PROGRAM AnalogConversion
VAR
	
	i					: INT := 1; //charger 1-8
	j					: INT := 1;  // section 1 - 4 
	k					: INT := 1;  // cap 1-10
	m					: INT := 1; //form cap 1-12

END_VAR

//Converting raw data into Voltage Reading (0-10V), (0.5-4.5V)   
//unfinish


//MCP Charger 
//Analog Input
FOR i := 1 TO 8 BY 1 DO
	
	MCP_IO.Charger[i].ChargerType_12kV := NOT MCP_IO.Charger[i].ChargerType_50kV;
	//50kV chargers feedback
	MCP_IO.Charger[i].voltageFeedback_norm := Norm_x (raw_input := INT_TO_REAL (MCP_IO.Charger[i].voltageFeedback_raw),
													x_max := 32767,
													x_min := 0);

	MCP_IO.Charger[i].voltageFeedback := (EngVal.Max_50kVChargerVoltage - EngVal.Min_50kVChargerVoltage) * ADC_10V(
																							normal_input := MCP_IO.Charger[i].voltageFeedback_norm,
																							x_max := 10,
																							x_min := 0);
												
	MCP_IO.Charger[i].currentFeedback_norm := Norm_x (raw_input := INT_TO_REAL (MCP_IO.Charger[i].currentFeedback_raw),
													x_max := 32767,
													x_min := 0);

	MCP_IO.Charger[i].currentFeedback := (EngVal.Max_50kVChargerCurrent - EngVal.Min_50kVChargerCurrent) * ADC_10V(
																							normal_input := MCP_IO.Charger[i].currentFeedback_norm,
																							x_max := 10,
																							x_min := 0);
	//12kV chargers ???
	
	
END_FOR;

//Analog Output
//voltageSP = Required Charge Voltage******************
FOR i := 1 TO 8 BY 1 DO
	
	//if 50kV config selected
	IF MCP_IO.Charger[i].ChargerType_50kV = TRUE THEN 
		//set limits of charger voltage input 
		IF MCP_IO.Charger[i].voltageSP >= REAL_TO_INT (EngVal.Max_50kVChargerVoltage) THEN
			MCP_IO.Charger[i].voltageSP := REAL_TO_INT (EngVal.Max_50kVChargerVoltage);
		END_IF;
		
	//prepare output signal for 50kV chargers.
		MCP_IO.Charger[i].voltageSP_norm := Norm_x (raw_input := INT_TO_REAL (MCP_IO.Charger[i].voltageSP), 
												x_max := EngVal.Max_50kVChargerVoltage,
												x_min := EngVal.Min_50kVChargerVoltage);	
												
		MCP_IO.Charger[i].voltageSP_raw := AQ (norm_input := MCP_IO.Charger[i].voltageSP_norm, 
												x_max := 10,
												x_min := 0);
		
	END_IF;
		
	//if 12kV config selected
	IF MCP_IO.Charger[i].ChargerType_12kV = TRUE THEN
		//set limits of charger voltage input 
		IF MCP_IO.Charger[i].voltageSP >= REAL_TO_INT (EngVal.Max_12kVChargerVoltage) THEN
			MCP_IO.Charger[i].voltageSP := REAL_TO_INT (EngVal.Max_12kVChargerVoltage);
		END_IF;
		
		
		//prepare output signal for 12kV chargers.
		MCP_IO.Charger[i].voltageSP_norm := Norm_x (raw_input := INT_TO_REAL (MCP_IO.Charger[i].voltageSP), 
												x_max := EngVal.Max_12kVChargerVoltage,
												x_min := EngVal.Min_12kVChargerVoltage);
		
		MCP_IO.Charger[i].voltageSP_raw := AQ (norm_input := MCP_IO.Charger[i].voltageSP_norm, 
												x_max := 10,
												x_min := 0); 
	END_IF;	
												
	//limite for output sigal (<= 10V)  this should not happen
	IF MCP_IO.Charger[i].voltageSP_raw >= 32767 THEN 
		MCP_IO.Charger[i].voltageSP_raw := 32767; 										
	END_IF;
	
END_FOR;

//prepare analog output for gls chargers.	
MCP_IO.GLS1_voltageSP_norm := Norm_x (raw_input := INT_TO_REAL (MCP_IO.GLS1_voltageSP),
									x_max := EngVal.Max_GLS1_ChargerV,
									x_min := 0);
MCP_IO.GLS1_voltageSP_raw:= AQ (norm_input := MCP_IO.GLS1_voltageSP_norm,
									x_max := 10,
									x_min := 0);									
									
MCP_IO.GLS2_voltageSP_norm := Norm_x (raw_input := INT_TO_REAL (MCP_IO.GLS2_voltageSP),
									x_max := EngVal.Max_GLS2_ChargerV,
									x_min := 0);
MCP_IO.GLS2_voltageSP_raw:= AQ (norm_input := MCP_IO.GLS2_voltageSP_norm,
									x_max := 10,
									x_min := 0);	

MCP_IO.GLS3_voltageSP_norm := Norm_x (raw_input := INT_TO_REAL (MCP_IO.GLS3_voltageSP),
									x_max := EngVal.Max_GLS3_ChargerV,
									x_min := 0);
MCP_IO.GLS3_voltageSP_raw:= AQ (norm_input := MCP_IO.GLS3_voltageSP_norm,
									x_max := 10,
									x_min := 0);	

//LCP 1 - 3 AI
FOR j := 1 TO 3 BY 1 DO 
	FOR k := 1 TO 10 BY 1 DO 
		LCP.Section[j].Peak.Cap[k].voltageFeedback_Norm := Norm_x (raw_input := INT_TO_REAL (LCP.Section[j].Peak.Cap[k].voltageFeedback_raw),
																x_max := 32767,
																x_min := 0);
																
		LCP.Section[j].Peak.Cap[k].voltageFeedback := (EngVal.Max_CapVoltage - EngVal.Min_CapVoltage) * ADC_10V (
																								normal_input := LCP.Section[j].Peak.Cap[k].voltageFeedback_Norm,
																								x_max := 10,
																								x_min := 0);
		//sustain caps 1 - 2
		LCP.Section[j].Sust.Cap[1].voltageFeedback_Norm := Norm_x (raw_input := INT_TO_REAL (LCP.Section[j].Sust.Cap[1].voltageFeedback_raw),
																x_max := 32767,
																x_min := 0);
																
		LCP.Section[j].Sust.Cap[1].voltageFeedback := (EngVal.Max_CapVoltage - EngVal.Min_CapVoltage) * ADC_10V (
																								normal_input := LCP.Section[j].Sust.Cap[1].voltageFeedback_Norm,
																								x_max := 10,
																								x_min := 0);
																
		LCP.Section[j].Sust.Cap[2].voltageFeedback_Norm := Norm_x (raw_input := INT_TO_REAL (LCP.Section[j].Sust.Cap[2].voltageFeedback_raw),
																x_max := 32767,
																x_min := 0);
																
		LCP.Section[j].Sust.Cap[2].voltageFeedback := (EngVal.Max_CapVoltage - EngVal.Min_CapVoltage) * ADC_10V (
																								normal_input := LCP.Section[j].Sust.Cap[2].voltageFeedback_Norm,
																								x_max := 10,
																								x_min := 0);
	END_FOR;	
END_FOR

//LCP 4 AI
FOR m := 1 TO 12 BY 1 DO
	LCP.Section[4].Form.Cap[m].voltageFeedback_norm := Norm_x (raw_input := INT_TO_REAL (LCP.Section[4].Form.Cap[m].voltageFeedback_raw),
																x_max := 32767,
																x_min := 0);
																
	LCP.Section[4].Form.Cap[m].voltageFeedback := (EngVal.Max_CapVoltage - EngVal.Min_CapVoltage) * ADC_10V (
																							normal_input := LCP.Section[4].Form.Cap[m].voltageFeedback_norm,
																							x_max := 10,
																							x_min := 0);
END_FOR;

//preform  cap AI
LCP.Section[4].PreFormCapVoltage_norm := Norm_x (raw_input := INT_TO_REAL (LCP.Section[4].PreFormCapVoltage_raw),
														x_max := 32767,
														x_min := 0);
															
LCP.Section[4].PreFormCapVoltageFeedback := (EngVal.Max_CapVoltage - EngVal.Min_CapVoltage) * ADC_10V (
																							normal_input := LCP.Section[4].PreFormCapVoltage_norm,
																							x_max := 10,
																							x_min := 0);															

		

(*
// Voltage feedback - 10V = Max voltage (102V)
Devices.Coil[1].ChargerVoltageFeedback_norm := Norm_x (raw_input := INT_TO_REAL(Devices.Coil[1].ChargeVoltageFeedback_raw),
										x_max := 32767,
										x_min := 0);
										
InstrumentReading.R2_01_CH00 := Devices.Coil[1].ChargerVoltageFeedback_norm * 10;

//Charger Voltage = (max voltage - min voltage) * measured_voltage / range(voltage)
Devices.Coil[1].ChargeVoltageFeedback := (Max_chargerVoltage - Min_chargerVoltage) * ADC_10V (normal_input := Devices.Coil[1].ChargerVoltageFeedback_norm,
																					x_max := 10,
																					x_min := 0);

//Current feedback - 4.5V = 600Amp????
Devices.Coil[1].CurrentFeedback_norm := Norm_x (raw_input := INT_TO_REAL(Devices.Coil[1].CurrentFeedback_raw),
								x_max := 32767*4.5/10,
								x_min := 0);
						
InstrumentReading.R2_01_CH01 := Devices.Coil[1].CurrentFeedback_norm * 4.5;

//Current feedback for each ultracap
Devices.Coil[1].CurrentFeedback := (Max_current_perCap - Min_current_perCap) * ADC_5V (normal_input := Devices.Coil[1].CurrentFeedback_norm,
																								x_max := 4.5,
																								x_min := 0.5);


																
//PWM Output

//set limits of charger voltage input 
FOR i := 1 TO 10 BY 1 DO
	IF Devices.Coil[i].chargerSetpoint >= REAL_TO_INT (Max_chargerVoltage) THEN
		Devices.Coil[i].chargerSetpoint := REAL_TO_INT (Max_chargerVoltage);
	END_IF;
	//This should never happend
	IF Devices.Coil[i].chargerSetpoint_raw >= (10/24 * 32767) THEN
		Devices.Coil[i].chargerSetpoint_raw := (10/24 * 32767);
	END_IF;
END_FOR;

Devices.Coil[1].chargerSetpoint_norm := Norm_x (raw_input := INT_TO_REAL (Devices.Coil[1].chargerSetpoint), 
												x_max := Max_chargerVoltage,
												x_min := Min_chargerVoltage);

Devices.Coil[1].chargerSetpoint_raw := PWMO (norm_input := Devices.Coil[1].chargerSetpoint_norm, 
												x_max := 24,
												x_min := 0); 	


//Current set point output
//set limits of charger voltage input 
FOR i := 1 TO 10 BY 1 DO
	IF Devices.Coil[i].currentSetpoint >= REAL_TO_INT (Max_current_perCap) THEN
		Devices.Coil[i].currentSetpoint := REAL_TO_INT (Max_current_perCap);
	END_IF;
	//This should never happend - Current setpoint board takes 0.5V - 4.5V
	IF Devices.Coil[i].currentSetpoint_raw >= (4.5/24 * 32767) THEN
		Devices.Coil[i].currentSetpoint_raw := (4.5/24 * 32767);
	END_IF;
END_FOR;

Devices.Coil[1].currentSetpoint_norm := Norm_x (raw_input := INT_TO_REAL (Devices.Coil[1].currentSetpoint), 
												x_max := Max_current_perCap,
												x_min := Min_current_perCap);
//current output for each cap
Devices.Coil[1].currentSetpoint_raw := PWMO (norm_input := Devices.Coil[1].currentSetpoint_norm, 
												x_max := 24,
												x_min := 0); 	


//uncomment this when PWM output module is ready.											
(*
//LCP1
Output.R2_02_00 := Devices.Coil[1].chargerSetpoint_raw; 
Output.R2_02_01 := Devices.Coil[1].currentSetpoint_raw;

//LCP2
Output.R3_02_00 := Devices.Coil[2].chargerSetpoint_raw; 
Output.R3_02_01 := Devices.Coil[2].currentSetpoint_raw;
*)

*)


//reset counter
IF i > 8 THEN
	i:=1;
END_IF;

IF j > 3 THEN 
	j := 1;
END_IF

IF k > 10 THEN 
	k := 1;
END_IF

IF m > 12 THEN 
	m := 1;
END_IF

END_PROGRAM

(* stored: Version 1.1.0.1, ProductVersion 3.1.4024.11
   POU AnalogConversion: Id {3b8eecca-a8e5-4cfd-bb8d-8865397a6f0b}, SpecialFunc None *)
